FUNCTION_BLOCK E_CALIBRATE_2P (* Event-driven two-point calibration (Low/High, independently stored - no EICO-before-EICS style ordering dependency) *)
  (* Standard: 61499-1 *)
  (* Version 1.0, 2026-09-11, Meisterschulen am Ostbahnhof, Ersatz fuer E_CALIBRATE_SQ: dieselbe Formel/dasselbe Ergebnis, aber ohne die EICO-vor-EICS-Abhaengigkeit - jeder Punkt speichert unabhaengig seinen Rohwert (wie E_CALIBRATE_3P), die Interpolation passiert erst live bei REQ, nicht mehr inkrementell beim Kalibrieren selbst. *)
  PACKAGE OSCAT::Basic::POUs::Engineering::measurements;
  (* Documentation:
  Formula
    Y = LOW_REF + (X - X_LOW) * (HIGH_REF - LOW_REF) / (X_HIGH - X_LOW) Why this replaces E_CALIBRATE_SQ
   E_CALIBRATE_SQ computes OFFSET/SCALE incrementally (EICO sets OFFSET from a live SCALE, EICS then recomputes both from an internal X_LOW_INT/Y_LOW_INT captured by EICO) - EICS is only mathematically valid after EICO has run at least once, which needed an ECC-enforced order to avoid a silent garbage-OFFSET calibration.
   This type stores X_LOW/X_HIGH completely independently (exactly like E_CALIBRATE_3P stores X_MIN/X_MID/X_MAX) and only combines them into a line at read-time (REQ), which runs regardless of calibration state. There is no data dependency between EI_LOW and EI_HIGH, so there is nothing an enforced order could protect against.
   Calibration (Two-Point, Free Order)
    - Low (EI_LOW): Apply low reference, set LOW_REF to desired output, fire EI_LOW → X_LOW := X
   - High (EI_HIGH): Apply high reference, set HIGH_REF to desired output, fire EI_HIGH → X_HIGH := X
    Either point can be recalibrated on its own at any later time without repeating the other.
   ECC State Machine
    START --REQ--> REQ --1--> START        (normal operation) START -EI_LOW-> C_LOW  --1--> START    (calibrate low point) START -EI_HIGH-> C_HIGH --1--> START   (calibrate high point) All calibration events are independently accessible from START - no enforced order.
  *)
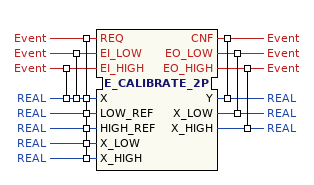
  EVENT_INPUT
    REQ WITH X, LOW_REF, HIGH_REF, X_LOW, X_HIGH; (* Normal Execution Request (berechnet Y) *)
    EI_LOW WITH X; (* Calibrate Low Point (speichert X_LOW := X) *)
    EI_HIGH WITH X; (* Calibrate High Point (speichert X_HIGH := X) *)
  END_EVENT
  EVENT_OUTPUT
    CNF WITH Y; (* Execution Confirmed *)
    EO_LOW WITH X_LOW; (* Low Point Calibrated *)
    EO_HIGH WITH X_HIGH; (* High Point Calibrated *)
  END_EVENT
  VAR_INPUT
    X : REAL; (* Raw input value *)
    LOW_REF : REAL; (* Target output Y at the low calibration point *)
    HIGH_REF : REAL; (* Target output Y at the high calibration point *)
  END_VAR
  VAR_OUTPUT
    Y : REAL; (* Calibrated output *)
  END_VAR
  VAR_IN_OUT
    X_LOW : REAL := 0.0; (* Stored raw value at the low calibration point *)
    X_HIGH : REAL := 1.0; (* Stored raw value at the high calibration point *)
  END_VAR
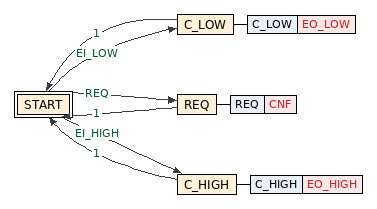
  EC_STATES
    START;
    REQ : REQ -> CNF;
    C_LOW : C_LOW -> EO_LOW;
    C_HIGH : C_HIGH -> EO_HIGH;
  END_STATES
  EC_TRANSITIONS
    START TO REQ := REQ;
    REQ TO START := 1;
    START TO C_LOW := EI_LOW;
    C_LOW TO START := 1;
    START TO C_HIGH := EI_HIGH;
    C_HIGH TO START := 1;
  END_TRANSITIONS
  ALGORITHM REQ IN ST:
(* live linear interpolation between the two independently stored points - no clipping, matching E_CALIBRATE_SQ's behaviour *)
IF (X_HIGH - X_LOW) <> 0.0 THEN
	Y := LOW_REF + (X - X_LOW) * (HIGH_REF - LOW_REF) / (X_HIGH - X_LOW);
ELSE
	Y := LOW_REF;
END_IF;
  END_ALGORITHM
  ALGORITHM C_LOW IN ST:
(* store current raw input as the low calibration point *)
X_LOW := X;
  END_ALGORITHM
  ALGORITHM C_HIGH IN ST:
(* store current raw input as the high calibration point *)
X_HIGH := X;
  END_ALGORITHM
END_FUNCTION_BLOCK
